(* IEC 61131-3 sources: RL_MAR/experiments/results/ablation/Ablation_single_agent_deepseek-ai_DeepSeek-V3.2_20260603_033757 (part 2) *)

(* ---- med_51.st ---- *)
FUNCTION_BLOCK PizzaMakingMachine
VAR_INPUT
    StartButton : BOOL;
    StopButton : BOOL;
    DoughReadySensor : BOOL;
    ToppingsReadySensor : BOOL;
    BakingDoneSensor : BOOL;
END_VAR

VAR_OUTPUT
    DoughRollerMotor : BOOL;
    ToppingDispenser : BOOL;
    ConveyorMotor : BOOL;
    OvenHeater : BOOL;
    OvenTemperature : INT;
END_VAR

VAR
    State : INT := 0; (* 0=Idle, 1=DoughRolling, 2=ToppingDispensing, 3=ConveyingToOven, 4=Baking, 5=Complete *)
    TargetBakingTemp : INT := 220;
    IdleTemp : INT := 0;
END_VAR

(* Main state machine *)
CASE State OF
    0: (* Idle State *)
        DoughRollerMotor := FALSE;
        ToppingDispenser := FALSE;
        ConveyorMotor := FALSE;
        OvenHeater := FALSE;
        OvenTemperature := IdleTemp;

        IF StartButton AND NOT StopButton THEN
            State := 1;
        END_IF;

    1: (* Dough Rolling State *)
        IF StopButton THEN
            State := 0;
        ELSE
            DoughRollerMotor := NOT DoughReadySensor;
            ToppingDispenser := FALSE;
            ConveyorMotor := FALSE;
            OvenHeater := FALSE;
            OvenTemperature := IdleTemp;

            IF DoughReadySensor THEN
                State := 2;
            END_IF;
        END_IF;

    2: (* Topping Dispensing State *)
        IF StopButton THEN
            State := 0;
        ELSE
            DoughRollerMotor := FALSE;
            ToppingDispenser := NOT ToppingsReadySensor;
            ConveyorMotor := FALSE;
            OvenHeater := FALSE;
            OvenTemperature := IdleTemp;

            IF ToppingsReadySensor THEN
                State := 3;
            END_IF;
        END_IF;

    3: (* Convey to Oven State *)
        IF StopButton THEN
            State := 0;
        ELSE
            DoughRollerMotor := FALSE;
            ToppingDispenser := FALSE;
            ConveyorMotor := TRUE;
            OvenHeater := TRUE;
            OvenTemperature := TargetBakingTemp;

            (* Transition to baking state - in real implementation would use timer/sensor *)
            State := 4;
        END_IF;

    4: (* Baking State *)
        IF StopButton THEN
            State := 0;
        ELSE
            DoughRollerMotor := FALSE;
            ToppingDispenser := FALSE;
            ConveyorMotor := FALSE;
            OvenHeater := TRUE;
            OvenTemperature := TargetBakingTemp;

            IF BakingDoneSensor THEN
                State := 5;
            END_IF;
        END_IF;

    5: (* Baking Complete State *)
        IF StopButton THEN
            State := 0;
        ELSE
            DoughRollerMotor := FALSE;
            ToppingDispenser := FALSE;
            ConveyorMotor := FALSE;
            OvenHeater := FALSE;
            OvenTemperature := IdleTemp;

            (* Return to idle after completion *)
            State := 0;
        END_IF;

    ELSE
        (* Error state - reset to idle *)
        State := 0;
        DoughRollerMotor := FALSE;
        ToppingDispenser := FALSE;
        ConveyorMotor := FALSE;
        OvenHeater := FALSE;
        OvenTemperature := IdleTemp;
END_CASE;
END_FUNCTION_BLOCK

(* ---- med_52.st ---- *)
FUNCTION_BLOCK TrafficManagementSystem
VAR_INPUT
    VehicleCount1 : INT;
    VehicleCount2 : INT;
    VehicleCount3 : INT;
    VehicleCount4 : INT;
END_VAR

VAR_OUTPUT
    TrafficLight1 : BOOL;
    TrafficLight2 : BOOL;
    TrafficLight3 : BOOL;
    TrafficLight4 : BOOL;
END_VAR

VAR
    // Internal variables to handle tie conditions and maintain state
    bDefaultStatePair1 : BOOL := TRUE;
    bDefaultStatePair2 : BOOL := TRUE;
END_VAR

(* Pair 1: Intersection 1 vs Intersection 2 - Independent Management *)
IF VehicleCount1 > VehicleCount2 THEN
    TrafficLight1 := TRUE;
    TrafficLight2 := FALSE;
    bDefaultStatePair1 := TRUE;  // Update default for next tie
ELSIF VehicleCount2 > VehicleCount1 THEN
    TrafficLight1 := FALSE;
    TrafficLight2 := TRUE;
    bDefaultStatePair1 := FALSE;  // Update default for next tie
ELSE
    (* If counts are equal, use alternating default logic *)
    TrafficLight1 := bDefaultStatePair1;
    TrafficLight2 := NOT bDefaultStatePair1;
    bDefaultStatePair1 := NOT bDefaultStatePair1;  // Toggle for next tie
END_IF;

(* Pair 2: Intersection 3 vs Intersection 4 - Independent Management *)
IF VehicleCount3 > VehicleCount4 THEN
    TrafficLight3 := TRUE;
    TrafficLight4 := FALSE;
    bDefaultStatePair2 := TRUE;  // Update default for next tie
ELSIF VehicleCount4 > VehicleCount3 THEN
    TrafficLight3 := FALSE;
    TrafficLight4 := TRUE;
    bDefaultStatePair2 := FALSE;  // Update default for next tie
ELSE
    (* If counts are equal, use alternating default logic *)
    TrafficLight3 := bDefaultStatePair2;
    TrafficLight4 := NOT bDefaultStatePair2;
    bDefaultStatePair2 := NOT bDefaultStatePair2;  // Toggle for next tie
END_IF;

END_FUNCTION_BLOCK

(* ---- med_53.st ---- *)
FUNCTION_BLOCK PouchMachine
VAR_INPUT
    start_machine: BOOL;
    stop_machine: BOOL;
    emergency_stop: BOOL := TRUE; (* Safety input - normally TRUE *)
    tension_sensor1: BOOL; (* Tension feedback from feeder 1 *)
    tension_sensor2: BOOL; (* Tension feedback from feeder 2 *)
    cutter_home_pos: BOOL; (* Horizontal cutter at home position *)
    cutter_vert_home: BOOL; (* Vertical cutter at home position *)
END_VAR

VAR_OUTPUT
    machine_ready: BOOL;
    feeder_running: BOOL;
    cutter_running: BOOL;
    heating_running: BOOL;
    cooling_running: BOOL;
    startup_in_progress: BOOL;
    shutdown_in_progress: BOOL;
    fault_condition: BOOL;
    fault_code: INT;
END_VAR

VAR
    startup_complete: BOOL := FALSE;
    shutdown_complete: BOOL := TRUE;
    machine_state: INT := 0;
    step_timer: TON;
    heating_stations_active: ARRAY[1..8] OF BOOL;
    cooling_stations_active: ARRAY[1..8] OF BOOL;
    feeder1_tension_ok: BOOL;
    feeder2_tension_ok: BOOL;
    winding_tension_ok: BOOL;
    horizontal_cutter_ready: BOOL;
    vertical_cutter_ready: BOOL;
    startup_step: INT := 0;
    shutdown_step: INT := 0;
    i: INT;
END_VAR

(* Initialize timers *)
step_timer(IN := FALSE, PT := T#1S);

(* Main state machine *)
IF emergency_stop THEN
    CASE machine_state OF
        (* IDLE STATE *)
        0: (* Machine stopped, ready for startup *)
            machine_ready := FALSE;
            feeder_running := FALSE;
            cutter_running := FALSE;
            heating_running := FALSE;
            cooling_running := FALSE;
            startup_in_progress := FALSE;
            shutdown_in_progress := FALSE;
            fault_condition := FALSE;
            fault_code := 0;
            startup_complete := FALSE;
            shutdown_complete := TRUE;

            (* Reset all stations *)
            FOR i := 1 TO 8 DO
                heating_stations_active[i] := FALSE;
                cooling_stations_active[i] := FALSE;
            END_FOR;

            horizontal_cutter_ready := FALSE;
            vertical_cutter_ready := FALSE;
            feeder1_tension_ok := FALSE;
            feeder2_tension_ok := FALSE;
            winding_tension_ok := FALSE;

            IF start_machine AND NOT stop_machine THEN
                machine_state := 1; (* Start startup sequence *)
                startup_step := 1;
                step_timer(IN := TRUE, PT := T#1S);
            END_IF;

        (* STARTUP SEQUENCE *)
        1: (* Startup sequence active *)
            startup_in_progress := TRUE;
            shutdown_in_progress := FALSE;

            CASE startup_step OF
                1: (* Step 1: Activate heating stations *)
                    heating_running := TRUE;
                    FOR i := 1 TO 8 DO
                        heating_stations_active[i] := TRUE;
                    END_FOR;

                    IF step_timer.Q THEN
                        step_timer(IN := FALSE, PT := T#1S);
                        startup_step := 2;
                        step_timer(IN := TRUE, PT := T#1S);
                    END_IF;

                2: (* Step 2: Activate cooling stations *)
                    cooling_running := TRUE;
                    FOR i := 1 TO 8 DO
                        cooling_stations_active[i] := TRUE;
                    END_FOR;

                    IF step_timer.Q THEN
                        step_timer(IN := FALSE, PT := T#1S);
                        startup_step := 3;
                        step_timer(IN := TRUE, PT := T#2S);
                    END_IF;

                3: (* Step 3: Start feeders and establish tension *)
                    feeder_running := TRUE;

                    (* Check tension from both feeders *)
                    feeder1_tension_ok := tension_sensor1;
                    feeder2_tension_ok := tension_sensor2;
                    winding_tension_ok := feeder1_tension_ok AND feeder2_tension_ok;

                    IF step_timer.Q THEN
                        IF winding_tension_ok THEN
                            step_timer(IN := FALSE, PT := T#1S);
                            startup_step := 4;
                            step_timer(IN := TRUE, PT := T#1S);
                        ELSE
                            (* Tension not established - fault *)
                            machine_state := 99;
                            fault_condition := TRUE;
                            fault_code := 1; (* Tension fault *)
                        END_IF;
                    END_IF;

                4: (* Step 4: Activate cutters *)
                    IF cutter_home_pos AND cutter_vert_home THEN
                        horizontal_cutter_ready := TRUE;
                        vertical_cutter_ready := TRUE;
                        cutter_running := TRUE;

                        IF step_timer.Q THEN
                            step_timer(IN := FALSE, PT := T#1S);
                            startup_step := 5;
                            step_timer(IN := TRUE, PT := T#500MS);
                        END_IF;
                    ELSE
                        (* Cutters not in home position - fault *)
                        machine_state := 99;
                        fault_condition := TRUE;
                        fault_code := 2; (* Cutter position fault *)
                    END_IF;

                5: (* Step 5: Set machine to ready state *)
                    IF step_timer.Q THEN
                        machine_ready := TRUE;
                        startup_complete := TRUE;
                        shutdown_complete := FALSE;
                        startup_in_progress := FALSE;
                        machine_state := 2; (* Running state *)
                        step_timer(IN := FALSE, PT := T#1S);
                    END_IF;
            END_CASE;

            (* Check for stop command during startup *)
            IF stop_machine THEN
                machine_state := 3; (* Go to shutdown *)
                shutdown_step := 1;
                step_timer(IN := TRUE, PT := T#1S);
            END_IF;

        (* RUNNING STATE *)
        2: (* Machine running normally *)
            (* Maintain station status *)
            heating_running := TRUE;
            cooling_running := TRUE;
            feeder_running := TRUE;
            cutter_running := TRUE;

            (* Continuously monitor tension *)
            feeder1_tension_ok := tension_sensor1;
            feeder2_tension_ok := tension_sensor2;
            winding_tension_ok := feeder1_tension_ok AND feeder2_tension_ok;

            IF NOT winding_tension_ok THEN
                machine_state := 99;
                fault_condition := TRUE;
                fault_code := 3; (* Running tension fault *)
            END_IF;

            (* Check for stop command *)
            IF stop_machine THEN
                machine_state := 3; (* Start shutdown sequence *)
                shutdown_step := 1;
                step_timer(IN := TRUE, PT := T#1S);
            END_IF;

        (* SHUTDOWN SEQUENCE *)
        3: (* Shutdown sequence active *)
            startup_in_progress := FALSE;
            shutdown_in_progress := TRUE;
            machine_ready := FALSE;

            CASE shutdown_step OF
                1: (* Step 1: Stop cutters *)
                    cutter_running := FALSE;
                    horizontal_cutter_ready := FALSE;
                    vertical_cutter_ready := FALSE;

                    IF step_timer.Q THEN
                        step_timer(IN := FALSE, PT := T#1S);
                        shutdown_step := 2;
                        step_timer(IN := TRUE, PT := T#1S);
                    END_IF;

                2: (* Step 2: Stop feeders *)
                    feeder_running := FALSE;
                    feeder1_tension_ok := FALSE;
                    feeder2_tension_ok := FALSE;
                    winding_tension_ok := FALSE;

                    IF step_timer.Q THEN
                        step_timer(IN := FALSE, PT := T#1S);
                        shutdown_step := 3;
                        step_timer(IN := TRUE, PT := T#2S);
                    END_IF;

                3: (* Step 3: Deactivate heating stations *)
                    heating_running := FALSE;
                    FOR i := 1 TO 8 DO
                        heating_stations_active[i] := FALSE;
                    END_FOR;

                    IF step_timer.Q THEN
                        step_timer(IN := FALSE, PT := T#1S);
                        shutdown_step := 4;
                        step_timer(IN := TRUE, PT := T#2S);
                    END_IF;

                4: (* Step 4: Deactivate cooling stations *)
                    cooling_running := FALSE;
                    FOR i := 1 TO 8 DO
                        cooling_stations_active[i] := FALSE;
                    END_FOR;

                    IF step_timer.Q THEN
                        step_timer(IN := FALSE, PT := T#1S);
                        shutdown_step := 5;
                        step_timer(IN := TRUE, PT := T#500MS);
                    END_IF;

                5: (* Step 5: Set machine to not-ready state *)
                    IF step_timer.Q THEN
                        startup_complete := FALSE;
                        shutdown_complete := TRUE;
                        shutdown_in_progress := FALSE;
                        machine_state := 0; (* Return to idle *)
                        step_timer(IN := FALSE, PT := T#1S);
                    END_IF;
            END_CASE;

            (* Check for start command during shutdown *)
            IF start_machine AND NOT stop_machine THEN
                (* Abort shutdown and restart *)
                machine_state := 1;
                startup_step := 1;
                step_timer(IN := TRUE, PT := T#1S);
            END_IF;

        (* FAULT STATE *)
        99: (* Fault condition *)
            machine_ready := FALSE;
            feeder_running := FALSE;
            cutter_running := FALSE;
            heating_running := FALSE;
            cooling_running := FALSE;
            startup_in_progress := FALSE;
            shutdown_in_progress := FALSE;

            (* Deactivate all stations *)
            FOR i := 1 TO 8 DO
                heating_stations_active[i] := FALSE;
                cooling_stations_active[i] := FALSE;
            END_FOR;

            (* Reset fault when emergency stop is cycled *)
            IF NOT emergency_stop THEN
                machine_state := 0;
                fault_condition := FALSE;
                fault_code := 0;
            END_IF;

    END_CASE;
ELSE
    (* Emergency stop active - force everything off *)
    machine_state := 0;
    machine_ready := FALSE;
    feeder_running := FALSE;
    cutter_running := FALSE;
    heating_running := FALSE;
    cooling_running := FALSE;
    startup_in_progress := FALSE;
    shutdown_in_progress := FALSE;
    fault_condition := FALSE;
    fault_code := 0;

    FOR i := 1 TO 8 DO
        heating_stations_active[i] := FALSE;
        cooling_stations_active[i] := FALSE;
    END_FOR;

    startup_complete := FALSE;
    shutdown_complete := TRUE;
    step_timer(IN := FALSE, PT := T#1S);
END_IF;
END_FUNCTION_BLOCK

(* ---- med_54.st ---- *)
FUNCTION_BLOCK FeedForwardControl
VAR_INPUT
    FlowRate1, FlowRate2: REAL; // Input flow rates of reactants
    MixRatio: REAL; // Desired mixing ratio (Reactant1:Reactant2)
END_VAR

VAR_OUTPUT
    OutFlowRate1, OutFlowRate2: REAL; // Output flow rates for reactants to maintain the mixing ratio
END_VAR

VAR
    MixedFlowRate: REAL; // Total mixed flow rate
    ClampedFlow1, ClampedFlow2: REAL;
    RatioPart1, RatioPart2: REAL;
    RatioSum: REAL;
END_VAR

// Limit input flow rates to allowed range 0-100
ClampedFlow1 := LIMIT(0.0, FlowRate1, 100.0);
ClampedFlow2 := LIMIT(0.0, FlowRate2, 100.0);

// Calculate total mixed flow rate
MixedFlowRate := ClampedFlow1 + ClampedFlow2;

// Calculate mixing ratio parts with error handling to prevent division by zero
RatioSum := MixRatio + 1.0;
IF RatioSum > 0.0 THEN
    RatioPart1 := MixRatio / RatioSum;
    RatioPart2 := 1.0 / RatioSum;
ELSE
    // Handle invalid ratio (MixRatio = -1.0)
    RatioPart1 := 0.0;
    RatioPart2 := 0.0;
END_IF

// Calculate output flow rates based on mixing ratio and total flow rate
OutFlowRate1 := LIMIT(0.0, MixedFlowRate * RatioPart1, 100.0);
OutFlowRate2 := LIMIT(0.0, MixedFlowRate * RatioPart2, 100.0);

END_FUNCTION_BLOCK

(* ---- med_55.st ---- *)
FUNCTION_BLOCK StateMachineControl
VAR_INPUT
    request : BOOL;
    done : BOOL;
END_VAR

VAR_OUTPUT
    listen : BOOL;
END_VAR

VAR
    state : INT := 0;
END_VAR

CASE state OF
    0: // Idle state
        listen := TRUE;
        IF request THEN
            state := 1;
            listen := FALSE;
        END_IF;

    1: // Processing state
        listen := FALSE;
        IF done THEN
            state := 0;
        END_IF;

    ELSE
        // Handle unexpected state values
        state := 0;
        listen := FALSE;
END_CASE;

END_FUNCTION_BLOCK

(* ---- med_56.st ---- *)
FUNCTION_BLOCK FB_SimpleRepeat
VAR_INPUT
    INPUT_VAR1 : INT := 2;
    INPUT_COUNTER : INT := 4;
END_VAR

VAR_OUTPUT
    OUTPUT_VAR1 : INT;
END_VAR

VAR
    COUNTER : INT;
END_VAR

METHOD Run : BOOL
VAR_INPUT
    bExecute : BOOL;
END_VAR

VAR
    nTempCounter : INT;
END_VAR

IF bExecute THEN
    OUTPUT_VAR1 := INPUT_VAR1;
    nTempCounter := INPUT_COUNTER;

    REPEAT
        OUTPUT_VAR1 := OUTPUT_VAR1 * 2;
        nTempCounter := nTempCounter - 1;
    UNTIL nTempCounter <= 0
    END_REPEAT;

    Run := TRUE;
ELSE
    Run := FALSE;
END_IF;

END_METHOD

END_FUNCTION_BLOCK

(* ---- med_57.st ---- *)
FUNCTION_BLOCK FB_CourseDifferenceControl
VAR_INPUT
    KOMPASS_GRAD : INT;
    KURS : INT;
END_VAR
VAR_OUTPUT
    KURS_DIFF : INT;
END_VAR
VAR
    tempDiff : INT;
END_VAR

// Main logic
IF KOMPASS_GRAD < 0 THEN
    KURS_DIFF := 0;
ELSE
    tempDiff := KURS - KOMPASS_GRAD;

    // Handle angle wrapping (3600 = 360 degrees * 10 for decimal precision)
    IF tempDiff > 1800 THEN
        tempDiff := tempDiff - 3600;
    ELSIF tempDiff < -1800 THEN
        tempDiff := tempDiff + 3600;
    END_IF;

    KURS_DIFF := tempDiff;
END_IF;
END_FUNCTION_BLOCK

PROGRAM MAIN
VAR
    courseControl : FB_CourseDifferenceControl;
    testKOMPASS : INT;
    testKURS : INT;
    resultDiff : INT;
END_VAR

// Example usage of the function block
courseControl(KOMPASS_GRAD := testKOMPASS, KURS := testKURS);
resultDiff := courseControl.KURS_DIFF;
END_PROGRAM

(* ---- med_58.st ---- *)
FUNCTION_BLOCK FB_ThresholdAccumulator
VAR_INPUT
    i : INT;
END_VAR

VAR_OUTPUT
    o : INT;
END_VAR

VAR
    s1 : INT;
END_VAR

// Main logic
s1 := 0; // Initialize s1 at start of each call

IF i > 0 THEN
    s1 := s1 + i; // Add i to s1 if i > 0
END_IF;

IF s1 = 42 THEN
    s1 := s1 + 8000; // Add 8000 if s1 equals 42
END_IF;

// Determine output value
IF s1 < 0 THEN
    o := 0;
ELSE
    o := s1;
END_IF;

END_FUNCTION_BLOCK

(* ---- med_59.st ---- *)
FUNCTION_BLOCK FB_ConditionalSelectAndAggregate
VAR_INPUT
    Z : INT;
END_VAR
VAR
    A_X : INT := 42;
    A_Y : INT := 333;
END_VAR
VAR_OUTPUT
    NEW_Z : INT;
END_VAR

IF A_X > Z THEN
    NEW_Z := A_Y;
ELSE
    NEW_Z := Z;
END_IF;
NEW_Z := NEW_Z + A_X + A_Y;
END_FUNCTION_BLOCK

(* ---- med_60.st ---- *)
FUNCTION_BLOCK FB_RequestHandler
VAR_INPUT
    request : BOOL;
    done : BOOL;
END_VAR

VAR_OUTPUT
    listen : BOOL;
END_VAR

VAR
    state : INT := 0;
END_VAR

CASE state OF
    0:
        IF NOT request THEN
            listen := TRUE;
            state := 0;
        ELSE
            listen := FALSE;
            state := 1;
        END_IF;

    1:
        IF NOT done THEN
            state := 1;
        ELSE
            listen := TRUE;
            state := 0;
        END_IF;
END_CASE;

END_FUNCTION_BLOCK

(* ---- med_61.st ---- *)
FUNCTION_BLOCK FB_Sum
VAR_INPUT
    maxValue : INT;
END_VAR
VAR_OUTPUT
    wData : WORD;
END_VAR

VAR
    II : INT;
END_VAR

BEGIN
    wData := 0;

    FOR II := 0 TO maxValue DO
        wData := wData + WORD(II);
    END_FOR;
END_FUNCTION_BLOCK

(* ---- med_62.st ---- *)
FUNCTION_BLOCK FB_PedestrianTrafficLight
VAR_INPUT
    pedBtnPress : BOOL;
END_VAR
VAR_OUTPUT
    carLightIsGreen : BOOL;
    pedLightIsGreen : BOOL;
    TimeCounter : INT;
END_VAR
VAR
    buttonPressedBefore : BOOL := FALSE;
    currentState : INT := 0; // 0: CarGreen, 1: CarRed_Waiting, 2: PedGreen, 3: PedRed_Waiting
END_VAR

CASE currentState OF
    0: // State 0: Car Green
        carLightIsGreen := TRUE;
        pedLightIsGreen := FALSE;
        TimeCounter := 0;

        // Check for button press transition
        IF (pedBtnPress AND NOT buttonPressedBefore) THEN
            currentState := 1;
            buttonPressedBefore := TRUE;
        ELSIF (pedBtnPress = FALSE) THEN
            buttonPressedBefore := FALSE;
        END_IF;

    1: // State 1: Car Red, Waiting for Pedestrian Green
        carLightIsGreen := FALSE;
        pedLightIsGreen := FALSE;
        TimeCounter := TimeCounter + 1;

        IF TimeCounter >= 10 THEN
            currentState := 2;
        END_IF;

        // Update button memory
        IF (pedBtnPress = FALSE) THEN
            buttonPressedBefore := FALSE;
        END_IF;

    2: // State 2: Pedestrian Green
        carLightIsGreen := FALSE;
        pedLightIsGreen := TRUE;
        TimeCounter := TimeCounter + 1;

        IF TimeCounter >= 40 THEN
            currentState := 3;
        END_IF;

        // Update button memory
        IF (pedBtnPress = FALSE) THEN
            buttonPressedBefore := FALSE;
        END_IF;

    3: // State 3: Pedestrian Red, Waiting for Car Green
        carLightIsGreen := FALSE;
        pedLightIsGreen := FALSE;
        TimeCounter := TimeCounter + 1;

        IF TimeCounter >= 50 THEN
            currentState := 0;
        END_IF;

        // Update button memory
        IF (pedBtnPress = FALSE) THEN
            buttonPressedBefore := FALSE;
        END_IF;
END_CASE;

END_FUNCTION_BLOCK

(* ---- med_63.st ---- *)
FUNCTION MoveCarToExitGate : BOOL
VAR_INPUT
    SpaceNumber : INT;
END_VAR
VAR
    // Add any necessary internal variables for movement logic
    // For example: Timer, Step counter, etc.
END_VAR

// Implement car movement logic here
// This is a placeholder - actual implementation would depend on hardware specifics
MoveCarToExitGate := TRUE; // Return TRUE when movement is complete
END_FUNCTION

FUNCTION_BLOCK Automated_Parking_Controller
VAR_INPUT
    EntryGateSensor : BOOL; (* Sensor input for entry gate *)
    ExitGateSensor : BOOL; (* Sensor input for exit gate *)
    CarDetected : BOOL; (* Sensor input for car detection *)
END_VAR
VAR_OUTPUT
    ParkingSpaceNumber : INT := 0; (* Allocated parking space number *)
    RetrievalInProgress : BOOL := FALSE; (* Flag for car retrieval in progress *)
END_VAR
VAR
    ParkingSpaces : ARRAY[1..100] OF BOOL; (* Parking space status: TRUE=Occupied, FALSE=Available *)
    i : INT; (* Loop counter *)
    SpaceToRetrieve : INT := 0; (* Parking space number for retrieval *)
    MovementComplete : BOOL; (* Flag to track movement completion *)
END_VAR

// Main program logic
IF NOT RetrievalInProgress THEN
    // Entry Gate Management
    IF EntryGateSensor THEN
        // Find first available parking space
        ParkingSpaceNumber := 0;
        FOR i := 1 TO 100 DO
            IF NOT ParkingSpaces[i] THEN
                ParkingSpaces[i] := TRUE;
                ParkingSpaceNumber := i;
                EXIT;
            END_IF;
        END_FOR;
    END_IF;

    // Exit Gate Management
    IF ExitGateSensor AND (ParkingSpaceNumber > 0) THEN
        ParkingSpaces[ParkingSpaceNumber] := FALSE;
        ParkingSpaceNumber := 0;
    END_IF;

    // Start car retrieval when detected
    IF CarDetected AND (ParkingSpaceNumber > 0) THEN
        RetrievalInProgress := TRUE;
        SpaceToRetrieve := ParkingSpaceNumber;
        MovementComplete := FALSE;
    END_IF;
END_IF;

// Car Retrieval Management
IF RetrievalInProgress THEN
    IF NOT MovementComplete THEN
        // Call the function (not instantiate it)
        MovementComplete := MoveCarToExitGate(SpaceToRetrieve);
    ELSE
        // Mark space as available and reset
        ParkingSpaces[SpaceToRetrieve] := FALSE;
        ParkingSpaceNumber := 0;
        RetrievalInProgress := FALSE;
        MovementComplete := FALSE;
        SpaceToRetrieve := 0;
    END_IF;
END_IF;
END_FUNCTION_BLOCK

(* ---- med_64.st ---- *)
FUNCTION_BLOCK BakeryOvenControl
VAR_INPUT
    TemperatureSensor : REAL;        (* Current measured oven temperature in °C *)
    HumiditySensor : REAL;           (* Current measured oven humidity in %RH *)
    StartBaking : BOOL;              (* Command to start baking cycle *)
    StopBaking : BOOL;               (* Command to stop baking cycle immediately *)
END_VAR

VAR_OUTPUT
    HeatingElement : BOOL;           (* Control signal for heating element *)
    CoolingElement : BOOL;           (* Control signal for cooling element *)
    HumidityControl : BOOL;          (* Control signal for humidification system *)
    DehumidityControl : BOOL;        (* Control signal for dehumidification system *)
    BakingComplete : BOOL;           (* Signal indicating baking cycle is complete *)
    RemainingTime : TIME;            (* Remaining baking time display *)
END_VAR

VAR
    (* Setpoints - initialized when oven is off *)
    TemperatureSetpoint : REAL := 180.0;     (* Desired baking temperature in °C *)
    HumiditySetpoint : REAL := 65.0;         (* Desired baking humidity in %RH *)
    BakingTimeSetpoint : TIME := T#30M;      (* Total baking time *)

    (* Control thresholds - configurable for different baking requirements *)
    TemperatureThreshold : REAL := 2.0;      (* Temperature deadband threshold *)
    HumidityThreshold : REAL := 5.0;         (* Humidity deadband threshold *)

    (* Internal state variables *)
    OvenActive : BOOL := FALSE;              (* TRUE when baking cycle is active *)
    TimerValue : TIME := T#0S;               (* Current timer value *)
    TimerEnable : BOOL := FALSE;             (* Timer enable flag *)

    (* Edge detection for start/stop commands *)
    StartRisingEdge : R_TRIG;
    StopRisingEdge : R_TRIG;
END_VAR

(* Edge detection for start/stop commands *)
StartRisingEdge(CLK := StartBaking);
StopRisingEdge(CLK := StopBaking);

(* Main control logic *)
IF NOT OvenActive THEN
    (* Oven is inactive - deactivate all outputs *)
    HeatingElement := FALSE;
    CoolingElement := FALSE;
    HumidityControl := FALSE;
    DehumidityControl := FALSE;
    BakingComplete := FALSE;
    TimerValue := T#0S;
    TimerEnable := FALSE;

    (* Initialize setpoints when oven is off (can be modified externally) *)
    TemperatureSetpoint := 180.0;    (* Default temperature setpoint *)
    HumiditySetpoint := 65.0;        (* Default humidity setpoint *)
    BakingTimeSetpoint := T#30M;     (* Default baking time *)

    (* Start baking cycle on rising edge of StartBaking *)
    IF StartRisingEdge.Q THEN
        OvenActive := TRUE;
        TimerValue := BakingTimeSetpoint;
        TimerEnable := TRUE;
        BakingComplete := FALSE;
    END_IF;

ELSE
    (* Oven is active - implement control logic *)

    (* Stop baking immediately if stop command received *)
    IF StopRisingEdge.Q THEN
        OvenActive := FALSE;
        HeatingElement := FALSE;
        CoolingElement := FALSE;
        HumidityControl := FALSE;
        DehumidityControl := FALSE;
        BakingComplete := TRUE;
        TimerEnable := FALSE;
    ELSE
        (* Temperature Control Logic *)
        IF TemperatureSensor < (TemperatureSetpoint - TemperatureThreshold) THEN
            (* Temperature below lower threshold - activate heating *)
            HeatingElement := TRUE;
            CoolingElement := FALSE;
        ELSIF TemperatureSensor > (TemperatureSetpoint + TemperatureThreshold) THEN
            (* Temperature above upper threshold - activate cooling *)
            HeatingElement := FALSE;
            CoolingElement := TRUE;
        ELSE
            (* Temperature within acceptable range - turn off both systems *)
            HeatingElement := FALSE;
            CoolingElement := FALSE;
        END_IF;

        (* Humidity Control Logic *)
        IF HumiditySensor < (HumiditySetpoint - HumidityThreshold) THEN
            (* Humidity below lower threshold - activate humidification *)
            HumidityControl := TRUE;
            DehumidityControl := FALSE;
        ELSIF HumiditySensor > (HumiditySetpoint + HumidityThreshold) THEN
            (* Humidity above upper threshold - activate dehumidification *)
            HumidityControl := FALSE;
            DehumidityControl := TRUE;
        ELSE
            (* Humidity within acceptable range - turn off both systems *)
            HumidityControl := FALSE;
            DehumidityControl := FALSE;
        END_IF;

        (* Baking Timer Logic *)
        IF TimerEnable AND (TimerValue > T#0S) THEN
            (* Decrement timer at one-second intervals *)
            TimerValue := TimerValue - T#1S;
        END_IF;

        (* Check if baking is complete *)
        IF TimerValue <= T#0S THEN
            (* Baking time elapsed - turn off all systems *)
            HeatingElement := FALSE;
            CoolingElement := FALSE;
            HumidityControl := FALSE;
            DehumidityControl := FALSE;
            BakingComplete := TRUE;
            TimerEnable := FALSE;
            OvenActive := FALSE;
        ELSE
            BakingComplete := FALSE;
        END_IF;
    END_IF;
END_IF;

(* Output remaining time for display *)
RemainingTime := TimerValue;

END_FUNCTION_BLOCK

(* ---- med_65.st ---- *)
FUNCTION_BLOCK TheaterControl
VAR_INPUT
    StartButton : BOOL;        (* Input for starting a performance *)
    StopButton : BOOL;         (* Input for stopping a performance *)
    SceneNumber : INT;         (* Input for selecting the scene or act *)
END_VAR
VAR_OUTPUT
    LightingControl : BOOL;    (* Output for controlling lighting *)
    SoundControl : BOOL;       (* Output for controlling sound *)
    PerformanceInProgress : BOOL; (* Indicator for an ongoing performance *)
END_VAR
VAR
    bStartRisingEdge : BOOL;   (* Edge detection for start button *)
    bPrevStartState : BOOL;    (* Previous state for edge detection *)
END_VAR

(* Edge detection for StartButton *)
bStartRisingEdge := StartButton AND NOT bPrevStartState;
bPrevStartState := StartButton;

(* Main control logic *)
IF StopButton THEN
    (* Immediate stop override *)
    LightingControl := FALSE;
    SoundControl := FALSE;
    PerformanceInProgress := FALSE;
ELSIF NOT PerformanceInProgress AND bStartRisingEdge THEN
    (* Start new performance if not already in progress *)
    IF (SceneNumber >= 1) AND (SceneNumber <= 3) THEN
        LightingControl := TRUE;
        SoundControl := TRUE;
        PerformanceInProgress := TRUE;
    ELSE
        (* Invalid scene number *)
        LightingControl := FALSE;
        SoundControl := FALSE;
        PerformanceInProgress := FALSE;
    END_IF;
ELSIF PerformanceInProgress THEN
    (* Maintain performance state *)
    IF (SceneNumber >= 1) AND (SceneNumber <= 3) THEN
        LightingControl := TRUE;
        SoundControl := TRUE;
        PerformanceInProgress := TRUE;
    ELSE
        (* Scene changed to invalid during performance - stop performance *)
        LightingControl := FALSE;
        SoundControl := FALSE;
        PerformanceInProgress := FALSE;
    END_IF;
ELSE
    (* Idle state - ensure outputs are off *)
    LightingControl := FALSE;
    SoundControl := FALSE;
    PerformanceInProgress := FALSE;
END_IF;
END_FUNCTION_BLOCK

(* ---- med_66.st ---- *)
FUNCTION_BLOCK ElevatorControl
VAR_INPUT
    CurrentPos : INT;
    RequestedPos : INT;
    ButtonPressed : BOOL;
END_VAR
VAR_OUTPUT
    MotorMovingUp : BOOL;
    MotorMovingDown : BOOL;
    DoorIsOpen : BOOL;
END_VAR
VAR
    bMoving : BOOL := FALSE;
END_VAR

(* Main elevator control logic *)
IF ButtonPressed THEN
    (* Close door when button is pressed *)
    DoorIsOpen := FALSE;

    (* Determine movement direction based on position comparison *)
    IF RequestedPos > CurrentPos THEN
        MotorMovingUp := TRUE;
        MotorMovingDown := FALSE;
        bMoving := TRUE;
    ELSIF RequestedPos < CurrentPos THEN
        MotorMovingUp := FALSE;
        MotorMovingDown := TRUE;
        bMoving := TRUE;
    ELSE
        (* Already at requested floor *)
        MotorMovingUp := FALSE;
        MotorMovingDown := FALSE;
        bMoving := FALSE;
        DoorIsOpen := TRUE;
    END_IF;
END_IF;

(* Stop and open door when reaching requested floor *)
IF CurrentPos = RequestedPos AND bMoving THEN
    MotorMovingUp := FALSE;
    MotorMovingDown := FALSE;
    bMoving := FALSE;
    DoorIsOpen := TRUE;
END_IF;

(* Ensure door remains closed while moving *)
IF bMoving THEN
    DoorIsOpen := FALSE;
END_IF;

(* Safety: Ensure motor cannot move in both directions simultaneously *)
IF MotorMovingUp AND MotorMovingDown THEN
    MotorMovingUp := FALSE;
    MotorMovingDown := FALSE;
    bMoving := FALSE;
END_IF;

END_FUNCTION_BLOCK

(* ---- med_67.st ---- *)
FUNCTION_BLOCK FB_FactorialCalculator
VAR_INPUT
    X : INT;
END_VAR

VAR_OUTPUT
    FactorialResult : INT;
    FactorialGoodResult : INT;
END_VAR

VAR
    tempGoodResult : INT;
END_VAR

// Initialize outputs
FactorialGoodResult := 0;
FactorialResult := 1;

// Check if input is within valid range
IF (X >= -3) AND (X <= 3) THEN
    // Calculate X^4 (X multiplied by itself 4 times)
    tempGoodResult := X * X * X * X;
    FactorialGoodResult := tempGoodResult;

    // Calculate FactorialResult based on FactorialGoodResult
    IF tempGoodResult > 1 THEN
        FactorialResult := tempGoodResult * (tempGoodResult - 1);
    ELSE
        FactorialResult := tempGoodResult;
    END_IF;
END_IF;

// If X is outside range [-3, 3], outputs remain at initialized values
// FactorialResult = 1 (as per overflow prevention requirement)
// FactorialGoodResult = 0
END_FUNCTION_BLOCK

(* ---- med_68.st ---- *)
FUNCTION_BLOCK FB_SignalControl
VAR_INPUT
    Int1 : BOOL;
    Int2 : BOOL;
    Int3 : BOOL;
    Int4 : BOOL;
    Int5 : BOOL;
    Int6 : BOOL;
    Int7 : BOOL;
    Int8 : BOOL;
    IntAn1 : UINT;
    IntAn2 : UINT;
    IntAn3 : UINT;
    IntAn4 : UINT;
    IntAn5 : UINT;
    IntAn6 : UINT;
    IntAn7 : UINT;
    IntAn8 : UINT;
    Marca2 : BOOL;
END_VAR

VAR_OUTPUT
    Out1 : BOOL;
    Out2 : BOOL;
    Out3 : BOOL;
    Out4 : BOOL;
    Out5 : BOOL;
    Out6 : BOOL;
    Out7 : BOOL;
    Out8 : BOOL;
    OutAn1 : UINT;
    OutAn2 : UINT;
    OutAn3 : UINT;
    OutAn4 : UINT;
    OutAn5 : UINT;
    OutAn6 : UINT;
    OutAn7 : UINT;
    OutAn8 : UINT;
END_VAR

VAR
    Marca1 : BOOL;
END_VAR

// Logic Implementation
// Marca1 and Marca2 latch logic
Marca1 := (NOT Marca2 AND (Marca1 OR NOT Out1) AND Int1) OR (Marca1 AND NOT Int1);
Marca2 := (NOT Marca1 AND (Marca2 OR Out1) AND Int1) OR (Marca2 AND NOT Int1);

// Out1 latch behavior
Out1 := (NOT Marca2 AND (Marca1 OR Out1)) OR (Out1 AND Marca2);

// Direct Boolean pass-through
Out2 := Int2;
Out3 := Int3;
Out4 := Int4;

// Direct unsigned integer pass-through
OutAn1 := IntAn1;
OutAn2 := IntAn2;
OutAn3 := IntAn3;
OutAn4 := IntAn4;

// Conditional output logic for Out5 to Out8
Out5 := (IntAn5 > 1000) AND NOT Int5;
Out6 := (IntAn6 > 1000) AND NOT Int6;
Out7 := (IntAn7 > 1000) AND NOT Int7;
Out8 := (IntAn8 > 1000) AND NOT Int8;

// Analog outputs pass-through for IntAn5 to IntAn8
OutAn5 := IntAn5;
OutAn6 := IntAn6;
OutAn7 := IntAn7;
OutAn8 := IntAn8;

END_FUNCTION_BLOCK

(* ---- med_69.st ---- *)
FUNCTION_BLOCK FB_ValueOut
VAR_INPUT
    valueIn : INT;
    conf : UINT;
END_VAR

VAR_OUTPUT
    ValueOut : INT;
END_VAR

VAR
END_VAR

METHOD ProcessValue : INT
VAR_INPUT
    valueIn : INT;
    conf : UINT;
END_VAR
VAR_OUTPUT
    result : INT;
END_VAR
BEGIN
    result := 0;

    CASE conf OF
        1, 2:
            IF valueIn <> 0 THEN
                result := valueIn / 10;
            END_IF;

        3:
            CASE valueIn OF
                0:   result := 0;
                300: result := 163;
                600: result := 331;
            ELSE
                result := 0;
            END_CASE;

        6, 7:
            IF valueIn = 100 THEN
                result := 319;
            ELSE
                result := 0;
            END_IF;

    ELSE
        result := 0;
    END_CASE;

    // Ensure non-negative output
    IF result < 0 THEN
        result := 0;
    END_IF;

    RETURN result;
END_METHOD

BEGIN
    ValueOut := ProcessValue(valueIn := valueIn, conf := conf);
END_FUNCTION_BLOCK

(* ---- med_70.st ---- *)
FUNCTION_BLOCK EggIncubatorControl
VAR_INPUT
    StartButton : BOOL;           (* Input for starting the incubation process *)
    StopButton : BOOL;            (* Input for stopping the incubation process *)
    TemperatureSensor : REAL;     (* Input for temperature reading in °C *)
    HumiditySensor : REAL;        (* Input for humidity reading in % *)
END_VAR
VAR_OUTPUT
    HeatingElement : BOOL;        (* Output for controlling the heating element *)
    Humidifier : BOOL;            (* Output for controlling the humidifier *)
    EggTurningMotor : BOOL;       (* Output for controlling the egg turning motor *)
    IncubationInProgress : BOOL;  (* Indicator for an ongoing incubation process *)
END_VAR
VAR
    TargetTemperature : REAL;     (* Target temperature in °C *)
    TargetHumidity : REAL;        (* Target humidity in % *)
    TurnIntervalSeconds : INT;    (* Interval for turning eggs (1 hour in seconds) *)
    TurnTimerSeconds : INT;       (* Timer for egg turning cycle in seconds *)
    MotorToggleFlag : BOOL;       (* Flag to track motor toggle state *)
END_VAR

(* Initialization of control parameters *)
TargetTemperature := 37.5;
TargetHumidity := 50.0;
TurnIntervalSeconds := 3600;

(* Start/Stop Control *)
IF StopButton THEN
    IncubationInProgress := FALSE;
    HeatingElement := FALSE;
    Humidifier := FALSE;
    EggTurningMotor := FALSE;
    TurnTimerSeconds := 0;
    MotorToggleFlag := FALSE;
ELSIF StartButton AND NOT IncubationInProgress THEN
    IncubationInProgress := TRUE;
    TurnTimerSeconds := 0;
    MotorToggleFlag := FALSE;
END_IF;

(* Temperature Control *)
IF IncubationInProgress THEN
    HeatingElement := (TemperatureSensor < TargetTemperature);
ELSE
    HeatingElement := FALSE;
END_IF;

(* Humidity Control *)
IF IncubationInProgress THEN
    Humidifier := (HumiditySensor < TargetHumidity);
ELSE
    Humidifier := FALSE;
END_IF;

(* Egg Turning Cycle *)
IF IncubationInProgress THEN
    TurnTimerSeconds := TurnTimerSeconds + 1;

    IF TurnTimerSeconds >= TurnIntervalSeconds THEN
        MotorToggleFlag := NOT MotorToggleFlag;
        EggTurningMotor := MotorToggleFlag;
        TurnTimerSeconds := 0;
    END_IF;
ELSE
    EggTurningMotor := FALSE;
    TurnTimerSeconds := 0;
END_IF;

END_FUNCTION_BLOCK

(* ---- med_71.st ---- *)
FUNCTION_BLOCK FB_Fibonacci_Calculator
VAR_INPUT
    N : DINT := 5;
END_VAR
VAR_OUTPUT
    O : DINT := 1;
END_VAR
VAR
    F1 : DINT := 1;
    F2 : DINT := 1;
    CNT : DINT := 2;
    Temp : DINT;
END_VAR

// Handle edge cases and calculate Fibonacci with saturation
IF N <= 0 THEN
    O := 0;
ELSIF N <= 2 THEN
    O := 1;
ELSE
    // Initialize Fibonacci sequence
    F1 := 1;
    F2 := 1;
    CNT := 2;

    // Calculate Fibonacci numbers up to N-th term
    WHILE CNT < N DO
        // Calculate next Fibonacci number with saturation check
        Temp := F1 + F2;

        // Apply saturation arithmetic - limit to INT maximum (32767)
        IF Temp > 32767 THEN
            Temp := 32767;
        END_IF;

        // Shift values for next iteration
        F1 := F2;
        F2 := Temp;

        // Increment counter
        CNT := CNT + 1;
    END_WHILE;

    // Output the N-th Fibonacci number
    O := F2;
END_IF;
END_FUNCTION_BLOCK

(* ---- med_72.st ---- *)
FUNCTION_BLOCK DigitalSignageManagement
VAR_INPUT
    DisplayLocations : ARRAY[1..10] OF BOOL;    (* Display status at each location *)
    ContentSource : ARRAY[1..10] OF INT;        (* Desired content for each location *)
END_VAR
VAR_OUTPUT
    CurrentContent : ARRAY[1..10] OF INT;       (* Current displayed content *)
END_VAR
VAR
    i : INT;                                    (* Loop counter *)
END_VAR

(* Main logic: Update content immediately based on inputs *)
FOR i := 1 TO 10 DO
    IF DisplayLocations[i] THEN
        (* Check if content code is valid (1, 2, or 3) *)
        CASE ContentSource[i] OF
            1: CurrentContent[i] := 1;    (* News *)
            2: CurrentContent[i] := 2;    (* Weather *)
            3: CurrentContent[i] := 3;    (* Promotional Content *)
        ELSE
            CurrentContent[i] := 0;       (* Invalid code or 0 = No Content *)
        END_CASE;
    ELSE
        (* Display is offline *)
        CurrentContent[i] := 0;
    END_IF;
END_FOR;

END_FUNCTION_BLOCK

(* ---- med_73.st ---- *)
FUNCTION_BLOCK RoboticWeldingSystem
VAR_INPUT
    RobotArm1Ready : BOOL;    (* Input for robot arm 1 ready status *)
    RobotArm2Ready : BOOL;    (* Input for robot arm 2 ready status *)
    WeldingGunReady : BOOL;   (* Input for welding gun ready status *)
    StartButton : BOOL;       (* Input for start button press *)
    StopButton : BOOL;        (* Input for stop button press *)
END_VAR
VAR_OUTPUT
    WeldingTrigger : BOOL;    (* Output to trigger welding *)
    WeldingComplete : BOOL;   (* Output indicating welding completion *)
END_VAR
VAR
    eState : (IDLE, WELDING); (* State variable for process control *)
END_VAR

(* Main state machine logic *)
CASE eState OF
    IDLE:
        WeldingTrigger := FALSE;
        WeldingComplete := TRUE;

        IF StopButton THEN
            (* Safety stop pressed - remain in IDLE *)
            eState := IDLE;
            WeldingComplete := TRUE;
        ELSIF RobotArm1Ready AND RobotArm2Ready AND WeldingGunReady AND StartButton THEN
            (* All conditions met - start welding *)
            eState := WELDING;
            WeldingComplete := FALSE;
        END_IF;

    WELDING:
        WeldingTrigger := TRUE;
        WeldingComplete := FALSE;

        IF StopButton THEN
            (* Safety stop pressed - abort welding *)
            eState := IDLE;
            WeldingTrigger := FALSE;
            WeldingComplete := TRUE;
        END_IF;
END_CASE;
END_FUNCTION_BLOCK

(* ---- med_74.st ---- *)
FUNCTION_BLOCK TrafficManagementSystem
VAR_INPUT
    VehicleCount1 : INT; (* Input for vehicle count at intersection 1 *)
    VehicleCount2 : INT; (* Input for vehicle count at intersection 2 *)
    VehicleCount3 : INT; (* Input for vehicle count at intersection 3 *)
    VehicleCount4 : INT; (* Input for vehicle count at intersection 4 *)
END_VAR
VAR_OUTPUT
    TrafficLight1 : BOOL; (* Output for traffic light at intersection 1 *)
    TrafficLight2 : BOOL; (* Output for traffic light at intersection 2 *)
    TrafficLight3 : BOOL; (* Output for traffic light at intersection 3 *)
    TrafficLight4 : BOOL; (* Output for traffic light at intersection 4 *)
END_VAR

(* Main logic *)
TrafficLight1 := (VehicleCount1 > VehicleCount2);
TrafficLight2 := NOT TrafficLight1;
TrafficLight3 := (VehicleCount3 > VehicleCount4);
TrafficLight4 := NOT TrafficLight3;

END_FUNCTION_BLOCK

(* ---- med_75.st ---- *)
FUNCTION_BLOCK HomeBrewingSystem
VAR_INPUT
    TemperatureSensor : REAL;      (* Current temperature in °C *)
    WaterFlowSensor : REAL;        (* Current water flow in L/min *)
    BrewingStartTime : TIME;       (* Start time of brewing process *)
    BrewingDuration : TIME;        (* Total brewing duration *)
END_VAR
VAR_OUTPUT
    HeatingElement : BOOL;         (* Control signal for heating element *)
    AgitationMotor : BOOL;         (* Control signal for agitation motor *)
    HopsDispenser : BOOL;          (* Control signal for hops dispenser *)
    FermentationTank : BOOL;       (* Control signal for fermentation tank transfer *)
END_VAR
VAR
    CurrentTime : TIME;            (* Current system time *)
    ElapsedBrewingTime : TIME;     (* Time elapsed since brewing start *)
    HopsDispensed : BOOL;          (* Flag to track if hops have been dispensed *)
    TankTransferred : BOOL;        (* Flag to track if transfer to fermentation tank occurred *)
END_VAR

(* Get current time *)
CurrentTime := TIME();

(* Calculate elapsed brewing time *)
ElapsedBrewingTime := CurrentTime - BrewingStartTime;

(* Temperature control logic *)
IF TemperatureSensor < 65.0 THEN
    HeatingElement := TRUE;
ELSE
    HeatingElement := FALSE;
END_IF;

(* Water flow control logic *)
IF WaterFlowSensor > 0.5 THEN
    AgitationMotor := TRUE;
ELSE
    AgitationMotor := FALSE;
END_IF;

(* Hops dispensing logic - dispense once after 5 hours *)
IF (ElapsedBrewingTime >= T#5h) AND (ElapsedBrewingTime <= BrewingDuration) AND NOT HopsDispensed THEN
    HopsDispenser := TRUE;
    HopsDispensed := TRUE;
ELSE
    HopsDispenser := FALSE;
END_IF;

(* Fermentation tank transfer logic - transfer once after 48 hours *)
IF (ElapsedBrewingTime >= T#48h) AND (ElapsedBrewingTime <= BrewingDuration) AND NOT TankTransferred THEN
    FermentationTank := TRUE;
    TankTransferred := TRUE;
ELSE
    FermentationTank := FALSE;
END_IF;

(* Reset flags when brewing duration is exceeded or before new brew starts *)
IF (ElapsedBrewingTime > BrewingDuration) OR (ElapsedBrewingTime < T#0s) THEN
    HopsDispensed := FALSE;
    TankTransferred := FALSE;
END_IF;

END_FUNCTION_BLOCK

(* ---- med_76.st ---- *)
FUNCTION_BLOCK MultimediaArtInstallationControl
VAR_INPUT
    MotionSensor : BOOL; (* Motion detection input *)
    AudioTrack : BOOL; (* Selected audio track *)
    VisualContent : BOOL; (* Selected visual content *)
END_VAR

VAR_OUTPUT
    LightingControl : BOOL; (* Lighting control output *)
    AudioControl : BOOL; (* Audio playback control *)
    VisualControl : BOOL; (* Visual display control *)
    ActivationTimer : INT; (* Timer for activation duration *)
END_VAR

VAR
    bMotionDetectedPrev : BOOL; (* Previous state of motion sensor for edge detection *)
    bElementsActive : BOOL; (* Flag indicating if elements are currently active *)
    tActivationTime : TIME; (* Activation time accumulator *)
    tNoMotionTime : TIME; (* No motion time accumulator *)
    bSafetyCheckOK : BOOL; (* Safety check status *)
END_VAR

VAR CONSTANT
    MAX_ACTIVATION_TIME : TIME := T#300S; (* Maximum activation time: 300 seconds *)
    DEBOUNCE_TIME : TIME := T#500MS; (* Debounce time for motion sensor *)
    SAFETY_CHECK_INTERVAL : TIME := T#10S; (* Interval for safety checks *)
END_VAR

(* Main control logic *)
IF NOT bSafetyCheckOK THEN
    (* Safety check failed - deactivate all elements *)
    LightingControl := FALSE;
    AudioControl := FALSE;
    VisualControl := FALSE;
    ActivationTimer := 0;
    tActivationTime := T#0S;
    tNoMotionTime := T#0S;
    bElementsActive := FALSE;
ELSE
    (* Edge detection for motion sensor with debouncing *)
    IF MotionSensor AND NOT bMotionDetectedPrev THEN
        (* Rising edge detected - start debounce timer *)
        tNoMotionTime := T#0S;
    ELSIF NOT MotionSensor AND bMotionDetectedPrev THEN
        (* Falling edge detected - start debounce timer *)
        tNoMotionTime := T#0S;
    END_IF;

    (* Update previous state *)
    bMotionDetectedPrev := MotionSensor;

    (* Check if motion is consistently detected for debounce time *)
    IF MotionSensor AND (tNoMotionTime >= DEBOUNCE_TIME) THEN
        (* Valid motion detected - activate elements *)
        IF NOT bElementsActive THEN
            (* Only activate if elements were not already active *)
            bElementsActive := TRUE;
            tActivationTime := T#0S;
        END_IF;
    ELSIF NOT MotionSensor AND (tNoMotionTime >= DEBOUNCE_TIME) THEN
        (* No motion detected for debounce time - deactivate elements *)
        bElementsActive := FALSE;
        tActivationTime := T#0S;
    END_IF;

    (* Control multimedia elements based on activation state and safety *)
    IF bElementsActive AND (tActivationTime < MAX_ACTIVATION_TIME) THEN
        (* Activate all elements *)
        LightingControl := TRUE;
        AudioControl := AudioTrack; (* Only activate if audio track is selected *)
        VisualControl := VisualContent; (* Only activate if visual content is selected *)

        (* Increment activation timer *)
        tActivationTime := tActivationTime + T#1S;
        ActivationTimer := TIME_TO_INT(tActivationTime);
    ELSE
        (* Deactivate all elements *)
        LightingControl := FALSE;
        AudioControl := FALSE;
        VisualControl := FALSE;

        (* Reset timer if elements are not active *)
        IF NOT bElementsActive THEN
            ActivationTimer := 0;
            tActivationTime := T#0S;
        END_IF;
    END_IF;

    (* Increment no motion timer when no motion is detected *)
    IF NOT MotionSensor THEN
        tNoMotionTime := tNoMotionTime + T#1S;
    ELSE
        tNoMotionTime := T#0S;
    END_IF;

    (* Safety protocol: Check power usage and system status *)
    (* This is a placeholder for actual safety checks *)
    bSafetyCheckOK := TRUE; (* Replace with actual safety logic *)

    (* Additional safety: Force deactivation if maximum time reached *)
    IF tActivationTime >= MAX_ACTIVATION_TIME THEN
        bElementsActive := FALSE;
        LightingControl := FALSE;
        AudioControl := FALSE;
        VisualControl := FALSE;
    END_IF;
END_IF;
END_FUNCTION_BLOCK

(* ---- med_77.st ---- *)
FUNCTION_BLOCK OutdoorLEDLightingControl
VAR_INPUT
    AmbientLight : REAL;    (* Ambient light sensor input in Lux *)
    MotionSensor : BOOL;    (* Motion sensor input *)
    EnergySaving : BOOL;    (* Energy saving mode switch *)
END_VAR

VAR_OUTPUT
    Light : BOOL;           (* LED lighting control output *)
    EnergyMode : BOOL;      (* Energy saving mode status output *)
END_VAR

(* Main control logic *)
IF MotionSensor THEN
    (* Motion Detection Override *)
    Light := TRUE;
    EnergyMode := FALSE;    (* Override energy-saving mode *)
ELSE
    (* No motion detected *)
    EnergyMode := EnergySaving;    (* Reflect energy saving input *)

    (* Ambient Light and Energy Saving Control *)
    IF (AmbientLight < 50.0) AND (NOT EnergySaving) THEN
        Light := TRUE;
    ELSE
        Light := FALSE;
    END_IF;
END_IF;

END_FUNCTION_BLOCK

(* ---- med_78.st ---- *)
FUNCTION_BLOCK RetractableRoofControl
VAR_INPUT
    RainSensor : BOOL;           (* TRUE if rain is detected *)
    WindSensor : BOOL;           (* TRUE if strong wind is detected *)
    TemperatureSensor : REAL;    (* Current temperature in degrees *)
END_VAR
VAR_OUTPUT
    RoofMotor : BOOL;            (* TRUE closes roof, FALSE opens roof *)
END_VAR

(* Main control logic *)
IF RainSensor AND WindSensor THEN
    (* Combined rain and wind - highest priority *)
    RoofMotor := TRUE;
ELSIF RainSensor THEN
    (* Rain only - medium priority *)
    RoofMotor := TRUE;
ELSIF TemperatureSensor < 20.0 THEN
    (* Low temperature - lowest priority *)
    RoofMotor := TRUE;
ELSE
    (* Normal conditions - open roof *)
    RoofMotor := FALSE;
END_IF;

END_FUNCTION_BLOCK

(* ---- med_79.st ---- *)
FUNCTION_BLOCK CapsuleFillingMachineControl
VAR_INPUT
    CapsuleWeight : REAL;           // Current capsule weight
    TargetWeight : REAL;            // Target weight to achieve
    CapsuleInPosition : BOOL;       // Capsule position sensor
    HopperEmpty : BOOL;             // Hopper empty sensor
END_VAR

VAR_OUTPUT
    FeederMotor : BOOL;             // Feeder motor control
    FillingMotor : BOOL;            // Filling motor control
    ConveyorMotor : BOOL;           // Conveyor motor control
    FillingInProgress : BOOL;       // Filling status
    ErrorCode : INT;                // Error code (0=No error)
END_VAR

VAR
    // State machine
    CurrentState : INT := 0;        // 0=IDLE, 1=CONVEYING, 2=FILLING, 3=CONVEYING_OUT
    PreviousState : INT := 0;

    // Timers
    ConveyorTimer : TON;
    FillingTimer : TON;
    ConveyOutTimer : TON;
    CapsuleDetectionTimer : TON;

    // PID controller variables (simplified implementation)
    PID_Kp : REAL := 0.5;           // Proportional gain
    PID_Ki : REAL := 0.1;           // Integral gain
    PID_Kd : REAL := 0.05;          // Derivative gain
    PID_Integral : REAL := 0.0;
    PID_PreviousError : REAL := 0.0;
    PID_LastTime : REAL := 0.0;
    PID_CycleTime : REAL := 0.1;    // 100ms cycle time
    PID_Output : REAL := 0.0;

    // Control variables
    WeightTolerance : REAL := 0.1;  // Tolerance for weight comparison
    ConveyorTimeSet : TIME := T#2S; // Conveyor operation time
    FillingTimeout : TIME := T#10S; // Maximum filling time
    ConveyOutTime : TIME := T#1S;   // Convey out time
    CapsuleDetectionTimeout : TIME := T#5S; // Timeout for capsule detection

    // Internal flags
    CapsuleDetected : BOOL := FALSE;
    FillingComplete : BOOL := FALSE;
    ConveyorStarted : BOOL := FALSE;

    // Error handling
    ErrorCapsuleTimeout : BOOL := FALSE;
    ErrorFillingTimeout : BOOL := FALSE;
    ErrorHopperLow : BOOL := FALSE;

    // Temporary variables
    CurrentTime : REAL;
    Error : REAL;
    Derivative : REAL;
    dt : REAL;
END_VAR

// Initialize outputs
FeederMotor := FALSE;
FillingMotor := FALSE;
ConveyorMotor := FALSE;
FillingInProgress := FALSE;
ErrorCode := 0;

// Safety Check - Hopper Empty
IF HopperEmpty THEN
    FeederMotor := FALSE;
    FillingMotor := FALSE;
    ConveyorMotor := FALSE;
    FillingInProgress := FALSE;
    ErrorCode := 1; // Hopper empty error
    CurrentState := 0; // Return to IDLE
    RETURN;
END_IF

// Weight Validation - Initial Check
IF CapsuleWeight >= TargetWeight - WeightTolerance THEN
    FeederMotor := FALSE;
    FillingMotor := FALSE;
    ConveyorMotor := FALSE;
    FillingInProgress := FALSE;
    CurrentState := 0; // Return to IDLE
    RETURN;
END_IF

// State Machine Implementation
CASE CurrentState OF
    0: // IDLE State
        FeederMotor := FALSE;
        FillingMotor := FALSE;
        ConveyorMotor := FALSE;
        FillingInProgress := FALSE;

        // Reset timers
        ConveyorTimer(IN:=FALSE, PT:=ConveyorTimeSet);
        FillingTimer(IN:=FALSE, PT:=FillingTimeout);
        ConveyOutTimer(IN:=FALSE, PT:=ConveyOutTime);
        CapsuleDetectionTimer(IN:=FALSE, PT:=CapsuleDetectionTimeout);

        // Reset flags
        CapsuleDetected := FALSE;
        FillingComplete := FALSE;
        ConveyorStarted := FALSE;
        ErrorCapsuleTimeout := FALSE;
        ErrorFillingTimeout := FALSE;

        // Reset PID controller
        PID_Integral := 0.0;
        PID_PreviousError := 0.0;
        PID_Output := 0.0;

        // Transition to CONVEYING when capsule is detected
        IF CapsuleInPosition THEN
            CurrentState := 1;
            CapsuleDetectionTimer(IN:=TRUE, PT:=CapsuleDetectionTimeout);
        END_IF

    1: // CONVEYING State
        ConveyorMotor := TRUE;
        ConveyorStarted := TRUE;
        FillingInProgress := FALSE;

        // Start conveyor timer
        ConveyorTimer(IN:=TRUE, PT:=ConveyorTimeSet);

        // Check for capsule detection timeout
        CapsuleDetectionTimer(IN:=TRUE, PT:=CapsuleDetectionTimeout);
        IF CapsuleDetectionTimer.Q THEN
            ErrorCapsuleTimeout := TRUE;
            ErrorCode := 2; // Capsule detection timeout
            CurrentState := 0; // Return to IDLE
        END_IF

        // Transition to FILLING after conveyor time or when weight indicates capsule is in position
        IF ConveyorTimer.Q OR (CapsuleWeight > 0.1) THEN
            CurrentState := 2;
            ConveyorMotor := FALSE;
            FillingInProgress := TRUE;
            PID_LastTime := REAL_TO_TIME(T#0ms) / 1000000.0; // Initialize time
        END_IF

    2: // FILLING State
        ConveyorMotor := FALSE;
        FillingInProgress := TRUE;

        // Start filling timer
        FillingTimer(IN:=TRUE, PT:=FillingTimeout);

        // Check for filling timeout
        IF FillingTimer.Q THEN
            ErrorFillingTimeout := TRUE;
            ErrorCode := 3; // Filling timeout
            CurrentState := 0; // Return to IDLE
            FillingMotor := FALSE;
        ELSE
            // Simplified PID Controller Implementation
            CurrentTime := REAL_TO_TIME(T#0ms) / 1000000.0; // Get current time in seconds

            // Calculate time difference
            dt := CurrentTime - PID_LastTime;
            IF dt < PID_CycleTime THEN
                // Wait for next cycle
                FillingMotor := FillingMotor; // Maintain current state
            ELSE
                // Calculate error
                Error := TargetWeight - CapsuleWeight;

                // Proportional term
                PID_Output := PID_Kp * Error;

                // Integral term (with anti-windup)
                IF ABS(Error) < TargetWeight * 0.5 THEN // Only integrate when error is reasonable
                    PID_Integral := PID_Integral + (PID_Ki * Error * dt);
                    // Limit integral term
                    IF PID_Integral > 100.0 THEN
                        PID_Integral := 100.0;
                    ELSIF PID_Integral < -100.0 THEN
                        PID_Integral := -100.0;
                    END_IF;
                END_IF;

                // Derivative term
                Derivative := PID_Kd * (Error - PID_PreviousError) / dt;

                // Calculate total output
                PID_Output := PID_Output + PID_Integral + Derivative;

                // Limit output to 0-100%
                IF PID_Output > 100.0 THEN
                    PID_Output := 100.0;
                ELSIF PID_Output < 0.0 THEN
                    PID_Output := 0.0;
                END_IF;

                // Control filling motor based on PID output
                FillingMotor := (PID_Output > 5.0); // Minimum 5% output to start motor

                // Update previous values
                PID_PreviousError := Error;
                PID_LastTime := CurrentTime;
            END_IF;

            // Check if target weight is reached
            IF CapsuleWeight >= TargetWeight - WeightTolerance THEN
                FillingMotor := FALSE;
                FillingComplete := TRUE;
                CurrentState := 3; // Transition to CONVEYING_OUT
                ConveyOutTimer(IN:=TRUE, PT:=ConveyOutTime);
            END_IF;
        END_IF;

    3: // CONVEYING_OUT State
        FillingMotor := FALSE;
        ConveyorMotor := TRUE;
        FillingInProgress := FALSE;

        // Start convey out timer
        ConveyOutTimer(IN:=TRUE, PT:=ConveyOutTime);

        // Transition back to IDLE after convey out time
        IF ConveyOutTimer.Q THEN
            ConveyorMotor := FALSE;
            CurrentState := 0;
        END_IF;

    ELSE
        // Default case - return to IDLE
        CurrentState := 0;
END_CASE;

// Update error code based on error flags
IF ErrorCapsuleTimeout THEN
    ErrorCode := 2;
ELSIF ErrorFillingTimeout THEN
    ErrorCode := 3;
ELSIF ErrorHopperLow THEN
    ErrorCode := 4;
END_IF;

// Update previous state
PreviousState := CurrentState;
END_FUNCTION_BLOCK

(* ---- med_80.st ---- *)
FUNCTION_BLOCK DoughMixerControl
VAR_INPUT
    IngredientsDetected : BOOL; (* Signal indicating presence of ingredients *)
END_VAR
VAR_OUTPUT
    MixingInProgress : BOOL; (* Control signal for mixer motor *)
END_VAR
VAR
    MixingTimeElapsed : TIME; (* Current elapsed mixing time *)
    MixingTimeLimit : TIME := T#5S; (* Configurable mixing time limit *)
    PrevIngredientsDetected : BOOL; (* Previous state for edge detection *)
END_VAR

(* Main control logic *)
IF IngredientsDetected AND NOT PrevIngredientsDetected THEN
    (* Rising edge detected - start new mixing cycle *)
    MixingTimeElapsed := T#0S;
    MixingInProgress := TRUE;
ELSIF NOT IngredientsDetected OR MixingTimeElapsed >= MixingTimeLimit THEN
    (* Stop mixing if ingredients removed or time limit reached *)
    MixingInProgress := FALSE;
END_IF

(* Timer increment logic - only while mixing is active *)
IF MixingInProgress THEN
    MixingTimeElapsed := MixingTimeElapsed + T#1S;
END_IF

(* Store current state for next cycle's edge detection *)
PrevIngredientsDetected := IngredientsDetected;
END_FUNCTION_BLOCK

(* ---- med_81.st ---- *)
FUNCTION_BLOCK SolarPanelTracking
VAR
    PanelAngle : REAL; (* Output for adjusting the solar panel angle *)
    SunriseTime : TIME := T#6H; (* Set the time for sunrise (6:00 AM) *)
    SunsetTime : TIME := T#18H; (* Set the time for sunset (6:00 PM) *)
    NoonTime : TIME := T#12H; (* Set the time for solar noon (12:00 PM) *)
    MorningAngle : REAL := 30.0; (* Set the morning angle for panels *)
    NoonAngle : REAL := 60.0; (* Set the noon angle for panels *)
    EveningAngle : REAL := 30.0; (* Set the evening angle for panels *)
END_VAR
VAR_INPUT
    CurrentTime : TIME;
    SolarIntensity : REAL;
END_VAR

(* Main execution logic *)
IF SolarIntensity >= 90.0 THEN
    PanelAngle := NoonAngle;
ELSE
    IF (CurrentTime < SunriseTime) OR (CurrentTime >= SunsetTime) THEN
        PanelAngle := 0.0;
    ELSIF (CurrentTime >= SunriseTime) AND (CurrentTime < NoonTime) THEN
        PanelAngle := MorningAngle;
    ELSIF (CurrentTime >= NoonTime) AND (CurrentTime < SunsetTime) THEN
        PanelAngle := EveningAngle;
    ELSE
        PanelAngle := 0.0; (* Fallback for any unhandled time condition *)
    END_IF;
END_IF;

END_FUNCTION_BLOCK

(* ---- med_82.st ---- *)
FUNCTION_BLOCK PetFeederControl
VAR_INPUT
    CurrentTime : TIME; (* Current system time input *)
END_VAR
VAR_OUTPUT
    FoodDispense : BOOL; (* Food dispenser control signal *)
END_VAR
VAR
    FeedTime1 : TIME := T#8H0M0S; (* First feeding time - 8:00 AM *)
    FeedTime2 : TIME := T#12H0M0S; (* Second feeding time - 12:00 PM *)
    FeedTime3 : TIME := T#18H0M0S; (* Third feeding time - 6:00 PM *)
    FoodAmount : INT := 50; (* Amount of food to dispense in grams - currently unused *)
END_VAR

(* Main dispensing logic *)
FoodDispense := FALSE;

IF (CurrentTime >= FeedTime1) AND (CurrentTime < (FeedTime1 + T#30S)) THEN
    FoodDispense := TRUE;
ELSIF (CurrentTime >= FeedTime2) AND (CurrentTime < (FeedTime2 + T#30S)) THEN
    FoodDispense := TRUE;
ELSIF (CurrentTime >= FeedTime3) AND (CurrentTime < (FeedTime3 + T#30S)) THEN
    FoodDispense := TRUE;
END_IF;

END_FUNCTION_BLOCK

(* ---- med_83.st ---- *)
FUNCTION_BLOCK AmusementRideControl
VAR_INPUT
    StartButton : BOOL;        (* Start button input *)
    StopButton : BOOL;         (* Emergency stop button input *)
    SpeedSensor : REAL;        (* Speed sensor input (RPM) *)
    SafetySensor : BOOL;       (* Safety sensor status *)
END_VAR
VAR_OUTPUT
    MotorOn : BOOL := FALSE;   (* Motor control output *)
    BrakeOn : BOOL := TRUE;    (* Brake control output *)
END_VAR
VAR
    SpeedLimit : REAL := 60.0; (* Maximum allowed speed in RPM *)
END_VAR

(* Emergency Stop - Highest Priority *)
IF StopButton THEN
    MotorOn := FALSE;
    BrakeOn := TRUE;
ELSE
    (* Start Condition - All Conditions Must Be Met *)
    IF StartButton AND
       (NOT StopButton) AND
       (SpeedSensor <= SpeedLimit) AND
       SafetySensor THEN
        MotorOn := TRUE;
        BrakeOn := FALSE;
    ELSE
        MotorOn := FALSE;
        BrakeOn := TRUE;
    END_IF;

    (* Normal Operation Monitoring - Continuous Check *)
    IF MotorOn AND
       ((SpeedSensor > SpeedLimit) OR (NOT SafetySensor)) THEN
        MotorOn := FALSE;
        BrakeOn := TRUE;
    END_IF;
END_IF;

END_FUNCTION_BLOCK

(* ---- med_84.st ---- *)
FUNCTION_BLOCK ParcelSortingSystem
VAR_INPUT
    ParcelSizeSensor : REAL;           (* Sensor input for parcel size in centimeters *)
    DestinationCodeSensor : INT;       (* Destination code: 1=Location A, 2=Location B *)
END_VAR

VAR_OUTPUT
    ConveyorBeltMotor : BOOL;          (* Output for conveyor belt motor: TRUE=On, FALSE=Off *)
    SortingGate1 : BOOL;               (* Output for sorting gate 1: TRUE=Open, FALSE=Closed *)
    SortingGate2 : BOOL;               (* Output for sorting gate 2: TRUE=Open, FALSE=Closed *)
END_VAR

VAR
    SizeThreshold : REAL := 50.0;      (* Threshold to distinguish large vs small parcels *)
    MinValidSize : REAL := 5.0;        (* Minimum valid parcel size to prevent false positives *)
    MaxValidSize : REAL := 200.0;      (* Maximum valid parcel size for system capacity *)
    ValidSizeDetected : BOOL;          (* Flag indicating if parcel size is within valid range *)
    ValidDestinationDetected : BOOL;   (* Flag indicating if destination code is valid *)
END_VAR

(* Main execution logic - runs on every PLC scan cycle *)

(* Validate sensor inputs *)
ValidSizeDetected := (ParcelSizeSensor >= MinValidSize) AND (ParcelSizeSensor <= MaxValidSize);
ValidDestinationDetected := (DestinationCodeSensor = 1) OR (DestinationCodeSensor = 2);

(* Control logic based on validated inputs *)
IF ValidSizeDetected AND ValidDestinationDetected THEN
    (* Valid parcel detected - activate conveyor belt *)
    ConveyorBeltMotor := TRUE;

    (* Sorting decision logic *)
    IF ParcelSizeSensor >= SizeThreshold THEN
        (* Large parcel: route to sorting gate 1 regardless of destination *)
        SortingGate1 := TRUE;
        SortingGate2 := FALSE;
    ELSIF DestinationCodeSensor = 1 THEN
        (* Small parcel destined for Location A: route to sorting gate 2 *)
        SortingGate1 := FALSE;
        SortingGate2 := TRUE;
    ELSE
        (* Small parcel destined for Location B: keep on main conveyor *)
        SortingGate1 := FALSE;
        SortingGate2 := FALSE;
    END_IF;
ELSE
    (* Invalid parcel detected: stop conveyor and close all gates for safety *)
    ConveyorBeltMotor := FALSE;
    SortingGate1 := FALSE;
    SortingGate2 := FALSE;
END_IF;

END_FUNCTION_BLOCK

(* ---- med_85.st ---- *)
FUNCTION_BLOCK ShredderControl
VAR_INPUT
    StartButton : BOOL;         (* Momentary start button *)
    StopButton : BOOL;          (* Momentary stop button *)
    EmergencyStop : BOOL;       (* Emergency stop button - active high *)
    MaterialInFeed : BOOL;      (* Sensor detecting material at infeed *)
    JammedSensor : BOOL;        (* Sensor detecting jam condition - active high *)
END_VAR
VAR_OUTPUT
    MotorControl : BOOL;        (* Control signal to motor starter *)
    SafetyRelay : BOOL;         (* Safety relay control *)
END_VAR
VAR
    bMotorRunning : BOOL;       (* Internal motor running state *)
    bSafetyCondition : BOOL;    (* Internal safety status *)
END_VAR

(* 1. Safety Logic - Highest Priority *)
(* Emergency stop OR jam detection deactivates safety *)
bSafetyCondition := NOT EmergencyStop AND NOT JammedSensor;
SafetyRelay := bSafetyCondition;

(* 2. Motor Control Logic *)
IF bSafetyCondition THEN
    (* Normal operation allowed *)

    (* Start conditions:
       1. Start button pressed (momentary)
       2. Material detected at infeed (auto-start) *)
    IF StartButton OR MaterialInFeed THEN
        bMotorRunning := TRUE;
    END_IF;

    (* Stop condition: Stop button pressed (momentary) *)
    IF StopButton THEN
        bMotorRunning := FALSE;
    END_IF;

    (* Apply motor command *)
    MotorControl := bMotorRunning;
ELSE
    (* Safety override: Emergency stop or jam detected *)
    MotorControl := FALSE;
    bMotorRunning := FALSE;
END_IF;

END_FUNCTION_BLOCK

(* ---- med_86.st ---- *)
FUNCTION_BLOCK FruitJuicingBottling
VAR_INPUT
    StartButton : BOOL;        (* Input for starting the process *)
    StopButton : BOOL;         (* Input for stopping the process *)
    FruitSelected : BOOL;      (* Input indicating fruit selection *)
END_VAR
VAR_OUTPUT
    JuiceProcessing : BOOL;    (* Output for controlling juice extraction *)
    BottleFilling : BOOL;      (* Output for controlling bottle filling *)
    CapPlacement : BOOL;       (* Output for placing caps on bottles *)
    Packaging : BOOL;          (* Output for packaging filled bottles *)
    ProcessInProgress : BOOL;  (* Indicator for an ongoing process *)
END_VAR
VAR
    eState : (IDLE, RUNNING);  (* State variable for process control *)
END_VAR

(* Main process logic *)
CASE eState OF
    IDLE:
        (* Reset all outputs when idle *)
        ProcessInProgress := FALSE;
        JuiceProcessing := FALSE;
        BottleFilling := FALSE;
        CapPlacement := FALSE;
        Packaging := FALSE;

        (* Check start conditions: StartButton pressed, fruit selected, and no process running *)
        IF StartButton AND FruitSelected AND NOT ProcessInProgress THEN
            eState := RUNNING;
        END_IF;

    RUNNING:
        (* Set process indicator and activate all concurrent stages *)
        ProcessInProgress := TRUE;
        JuiceProcessing := TRUE;
        BottleFilling := TRUE;
        CapPlacement := TRUE;
        Packaging := TRUE;

        (* Check stop conditions: StopButton pressed OR fruit deselected *)
        IF StopButton OR NOT FruitSelected THEN
            eState := IDLE;
        END_IF;
END_CASE;
END_FUNCTION_BLOCK

(* ---- med_87.st ---- *)
FUNCTION_BLOCK WaterDesalination
VAR_INPUT
    StartButton : BOOL;          (* Input for starting the desalination process *)
    StopButton : BOOL;           (* Input for stopping the desalination process *)
    SalinitySensor : REAL;       (* Input for salinity level measurement *)
END_VAR
VAR_OUTPUT
    SeawaterInletValve : BOOL;   (* Output for seawater inlet valve control *)
    FreshwaterOutletValve : BOOL; (* Output for freshwater outlet valve control *)
    DesalinationInProgress : BOOL; (* Indicator for an ongoing desalination process *)
END_VAR
VAR
    MaxSalinity : REAL := 35.0;  (* Maximum allowable salinity in ppm for freshwater *)
    SalinityControlSeconds : INT := 0; (* Timer for salinity control in seconds *)
END_VAR

(* Main logic *)
IF StopButton THEN
    (* Stop process immediately when StopButton is pressed *)
    DesalinationInProgress := FALSE;
    SeawaterInletValve := FALSE;
    FreshwaterOutletValve := FALSE;
    SalinityControlSeconds := 0;
ELSIF StartButton AND NOT DesalinationInProgress THEN
    (* Start process when StartButton is pressed and process is not already running *)
    DesalinationInProgress := TRUE;
    SeawaterInletValve := TRUE;
    FreshwaterOutletValve := TRUE;
    SalinityControlSeconds := 0;
END_IF;

(* Salinity monitoring and control *)
IF DesalinationInProgress THEN
    (* Increment timer each scan cycle - assuming 1 second per cycle *)
    SalinityControlSeconds := SalinityControlSeconds + 1;

    (* Check salinity every 10 seconds *)
    IF SalinityControlSeconds >= 10 THEN
        IF SalinitySensor > MaxSalinity THEN
            (* Close freshwater outlet valve if salinity is too high *)
            FreshwaterOutletValve := FALSE;
        ELSE
            (* Keep freshwater outlet valve open if salinity is acceptable *)
            FreshwaterOutletValve := TRUE;
        END_IF;
        (* Reset timer after check *)
        SalinityControlSeconds := 0;
    END_IF;
END_IF;

END_FUNCTION_BLOCK

(* ---- med_88.st ---- *)
FUNCTION_BLOCK SmartLockerControl
VAR_INPUT
    AccessCode : INT;     (* User entered access code *)
    LockerNumber : INT;   (* Selected locker number (1-10) *)
END_VAR
VAR_OUTPUT
    LockerOpen : BOOL;    (* TRUE when locker should open *)
END_VAR
VAR
    LockerStatus : ARRAY[1..10] OF BOOL;      (* TRUE=occupied/locked, FALSE=empty/unlocked *)
    LockerAccessCode : ARRAY[1..10] OF INT;   (* Unique access codes for each locker *)
    bInitDone : BOOL;                         (* Initialization flag *)
    i : INT;                                  (* Loop counter for initialization *)
END_VAR

(* Initialization - runs only once *)
IF NOT bInitDone THEN
    (* Initialize all lockers to occupied/locked (TRUE) *)
    FOR i := 1 TO 10 DO
        LockerStatus[i] := TRUE;
    END_FOR;

    (* Set individual access codes for each locker *)
    LockerAccessCode[1] := 1234;
    LockerAccessCode[2] := 5678;
    LockerAccessCode[3] := 9876;
    LockerAccessCode[4] := 4321;
    LockerAccessCode[5] := 6543;
    LockerAccessCode[6] := 7890;
    LockerAccessCode[7] := 3456;
    LockerAccessCode[8] := 8765;
    LockerAccessCode[9] := 2345;
    LockerAccessCode[10] := 6789;

    bInitDone := TRUE;
END_IF;

(* Default output state *)
LockerOpen := FALSE;

(* Access control logic *)
IF (LockerNumber >= 1) AND (LockerNumber <= 10) THEN
    (* Check if access code matches and locker is currently locked *)
    IF (AccessCode = LockerAccessCode[LockerNumber]) AND LockerStatus[LockerNumber] THEN
        LockerOpen := TRUE;               (* Open the locker *)
        LockerStatus[LockerNumber] := FALSE; (* Mark as empty/unlocked *)
    END_IF;
END_IF;
END_FUNCTION_BLOCK

(* ---- med_89.st ---- *)
FUNCTION_BLOCK SoilTestingDeviceControl
VAR_INPUT
    StartButton : BOOL;           (* Input for starting the testing process *)
    SoilSampleDetected : BOOL;    (* Input for detecting soil sample *)
END_VAR

VAR_OUTPUT
    NutrientPump : BOOL;          (* Output to control nutrient pump *)
    pHAdjustmentPump : BOOL;      (* Output to control pH adjustment pump *)
END_VAR

VAR
    pHSensorValue : REAL;         (* Simulated pH sensor value *)
    NutrientSensorValue : REAL;   (* Simulated nutrient sensor value *)
    TestingStatus : INT;          (* Status: 0=Idle, 1=Testing, 2=Completed *)
    NutrientThreshold : REAL := 0.7;   (* Nutrient level threshold for analysis *)
    pHThreshold : REAL := 6.5;         (* pH level threshold for analysis *)
END_VAR

(* Main logic implementation *)
CASE TestingStatus OF
    0: (* Idle state *)
        (* Initialize sensor values *)
        pHSensorValue := 7.0;
        NutrientSensorValue := 0.5;

        (* Ensure pumps are off in idle state *)
        NutrientPump := FALSE;
        pHAdjustmentPump := FALSE;

        (* Check for start command *)
        IF StartButton THEN
            TestingStatus := 1;
            NutrientPump := TRUE;
            pHAdjustmentPump := TRUE;
        END_IF;

    1: (* Testing state *)
        (* Update simulated sensor values during testing *)
        IF NutrientSensorValue < 0.9 THEN
            NutrientSensorValue := NutrientSensorValue + 0.1;
        END_IF;

        IF pHSensorValue > 4.0 THEN
            pHSensorValue := pHSensorValue - 0.5;
        END_IF;

        (* Check for sample detection and analysis *)
        IF SoilSampleDetected THEN
            IF (NutrientSensorValue >= NutrientThreshold) AND (pHSensorValue <= pHThreshold) THEN
                TestingStatus := 2;
                NutrientPump := FALSE;
                pHAdjustmentPump := FALSE;
            END_IF;
        END_IF;

    2: (* Completed state *)
        (* Ensure pumps are off when testing is completed *)
        NutrientPump := FALSE;
        pHAdjustmentPump := FALSE;

        (* Optionally, the system could be reset to idle here if needed *)
        (* TestingStatus := 0; *)  (* Uncomment if automatic reset is desired *)
END_CASE;

END_FUNCTION_BLOCK

(* ---- med_90.st ---- *)
FUNCTION_BLOCK SushiConveyorControl
VAR_INPUT
    StartButton : BOOL;     (* Input to start the conveyor *)
    StopButton : BOOL;      (* Input to stop the conveyor *)
    EmergencyStop : BOOL;   (* Input for emergency stop *)
END_VAR
VAR_OUTPUT
    ConveyorMotor : BOOL;   (* Output to control the conveyor motor *)
END_VAR
VAR
    BeltRunning : BOOL;     (* Status of the conveyor: Running or Stopped *)
    ConveyorTimer : INT;    (* Timer counter for conveyor rotation *)
    RotationTime : INT := 5; (* Time for one rotation in seconds *)
END_VAR

(* Emergency Stop - Highest Priority *)
IF EmergencyStop THEN
    ConveyorMotor := FALSE;
    BeltRunning := FALSE;
    ConveyorTimer := 0;
    RETURN;
END_IF;

(* Start/Stop Control *)
IF StartButton AND NOT BeltRunning THEN
    ConveyorMotor := TRUE;
    BeltRunning := TRUE;
    ConveyorTimer := 0;
ELSIF StopButton AND BeltRunning THEN
    ConveyorMotor := FALSE;
    BeltRunning := FALSE;
    ConveyorTimer := 0;
END_IF;

(* Simulated Rotation Cycle *)
IF BeltRunning THEN
    ConveyorTimer := ConveyorTimer + 1;
    IF ConveyorTimer >= RotationTime THEN
        ConveyorTimer := 0;
    END_IF;
    ConveyorMotor := TRUE;
END_IF;

END_FUNCTION_BLOCK

(* ---- med_91.st ---- *)
FUNCTION_BLOCK AGVControlSystem
VAR_INPUT
    MaterialRequest : INT; (* 新的物料请求，>0表示有效请求 *)
    TaskComplete_AGV1 : BOOL := FALSE; (* AGV1任务完成信号 *)
    TaskComplete_AGV2 : BOOL := FALSE; (* AGV2任务完成信号 *)
    TaskComplete_AGV3 : BOOL := FALSE; (* AGV3任务完成信号 *)
    AGV1_PositionUpdate : INT := 0; (* AGV1位置更新值 *)
    AGV2_PositionUpdate : INT := 0; (* AGV2位置更新值 *)
    AGV3_PositionUpdate : INT := 0; (* AGV3位置更新值 *)
END_VAR

VAR_OUTPUT
    AGV1_Ready : BOOL := TRUE; (* AGV1就绪状态 *)
    AGV2_Ready : BOOL := TRUE; (* AGV2就绪状态 *)
    AGV3_Ready : BOOL := TRUE; (* AGV3就绪状态 *)
    AGV1_CurrentTask : INT := 0; (* AGV1当前任务，0表示空闲 *)
    AGV2_CurrentTask : INT := 0; (* AGV2当前任务，0表示空闲 *)
    AGV3_CurrentTask : INT := 0; (* AGV3当前任务，0表示空闲 *)
    AGV1_Position : INT := 0; (* AGV1当前位置 *)
    AGV2_Position : INT := 0; (* AGV2当前位置 *)
    AGV3_Position : INT := 0; (* AGV3当前位置 *)
    QueueCount : INT := 0; (* 队列中任务数量 *)
    SafetyError : BOOL := FALSE; (* 安全错误标志 *)
    QueueOverflow : BOOL := FALSE; (* 队列溢出标志 *)
    InvalidRequest : BOOL := FALSE; (* 无效请求标志 *)
END_VAR

VAR
    (* 物料处理请求队列 - FIFO实现 *)
    MaterialQueue : ARRAY[1..10] OF INT;
    QueueHead : INT := 1; (* 队列头部指针 *)
    QueueTail : INT := 1; (* 队列尾部指针 *)

    (* AGV状态管理 *)
    AGVStatus : ARRAY[1..3] OF BOOL := [TRUE, TRUE, TRUE]; (* TRUE=就绪，FALSE=工作中 *)
    AGVTask : ARRAY[1..3] OF INT := [0, 0, 0]; (* AGV当前任务 *)

    (* 临时变量 *)
    TempTask : INT;
    i : INT;

    (* 状态监控 *)
    PreviousQueueCount : INT := 0;
    SystemIdle : BOOL := TRUE;
END_VAR

(* 1. 处理新的物料请求 *)
InvalidRequest := FALSE;
IF MaterialRequest > 0 THEN
    (* 检查请求有效性 *)
    IF MaterialRequest <= 100 THEN  (* 假设有效任务ID范围1-100 *)
        IF QueueCount < 10 THEN
            (* 原子性队列更新 *)
            MaterialQueue[QueueTail] := MaterialRequest;
            QueueTail := QueueTail + 1;
            IF QueueTail > 10 THEN
                QueueTail := 1;
            END_IF;
            QueueCount := QueueCount + 1;
            QueueOverflow := FALSE;
        ELSE
            (* 队列溢出处理 *)
            QueueOverflow := TRUE;
            SafetyError := TRUE;
        END_IF;
    ELSE
        (* 无效请求处理 *)
        InvalidRequest := TRUE;
        SafetyError := TRUE;
    END_IF;
END_IF;

(* 2. 处理AGV任务完成 *)
(* AGV1任务完成处理 *)
IF TaskComplete_AGV1 AND NOT AGVStatus[1] THEN
    AGVStatus[1] := TRUE;
    AGVTask[1] := 0;
    AGV1_Position := 0; (* 重置位置 *)
END_IF;

(* AGV2任务完成处理 *)
IF TaskComplete_AGV2 AND NOT AGVStatus[2] THEN
    AGVStatus[2] := TRUE;
    AGVTask[2] := 0;
    AGV2_Position := 0; (* 重置位置 *)
END_IF;

(* AGV3任务完成处理 *)
IF TaskComplete_AGV3 AND NOT AGVStatus[3] THEN
    AGVStatus[3] := TRUE;
    AGVTask[3] := 0;
    AGV3_Position := 0; (* 重置位置 *)
END_IF;

(* 3. 优先级任务分配策略 *)
IF QueueCount > 0 THEN
    (* 从队列头部获取任务 *)
    TempTask := MaterialQueue[QueueHead];

    (* 优先级分配：AGV1 > AGV2 > AGV3 *)
    IF AGVStatus[1] THEN
        (* 分配任务给AGV1 *)
        AGVTask[1] := TempTask;
        AGVStatus[1] := FALSE;

        (* 更新队列 *)
        QueueHead := QueueHead + 1;
        IF QueueHead > 10 THEN
            QueueHead := 1;
        END_IF;
        QueueCount := QueueCount - 1;

    ELSIF AGVStatus[2] THEN
        (* 分配任务给AGV2 *)
        AGVTask[2] := TempTask;
        AGVStatus[2] := FALSE;

        (* 更新队列 *)
        QueueHead := QueueHead + 1;
        IF QueueHead > 10 THEN
            QueueHead := 1;
        END_IF;
        QueueCount := QueueCount - 1;

    ELSIF AGVStatus[3] THEN
        (* 分配任务给AGV3 *)
        AGVTask[3] := TempTask;
        AGVStatus[3] := FALSE;

        (* 更新队列 *)
        QueueHead := QueueHead + 1;
        IF QueueHead > 10 THEN
            QueueHead := 1;
        END_IF;
        QueueCount := QueueCount - 1;
    END_IF;
END_IF;

(* 4. 更新AGV位置并实施安全约束 *)
(* AGV1位置更新 *)
IF NOT AGVStatus[1] THEN
    AGV1_Position := AGV1_Position + AGV1_PositionUpdate;
    (* 安全约束：确保位置非负 *)
    IF AGV1_Position < 0 THEN
        AGV1_Position := 0;
        SafetyError := TRUE;
    END_IF;
END_IF;

(* AGV2位置更新 *)
IF NOT AGVStatus[2] THEN
    AGV2_Position := AGV2_Position + AGV2_PositionUpdate;
    (* 安全约束：确保位置非负 *)
    IF AGV2_Position < 0 THEN
        AGV2_Position := 0;
        SafetyError := TRUE;
    END_IF;
END_IF;

(* AGV3位置更新 *)
IF NOT AGVStatus[3] THEN
    AGV3_Position := AGV3_Position + AGV3_PositionUpdate;
    (* 安全约束：确保位置非负 *)
    IF AGV3_Position < 0 THEN
        AGV3_Position := 0;
        SafetyError := TRUE;
    END_IF;
END_IF;

(* 5. 状态监控和同步 *)
(* 更新输出状态 *)
AGV1_Ready := AGVStatus[1];
AGV2_Ready := AGVStatus[2];
AGV3_Ready := AGVStatus[3];

AGV1_CurrentTask := AGVTask[1];
AGV2_CurrentTask := AGVTask[2];
AGV3_CurrentTask := AGVTask[3];

(* 监控系统空闲状态 *)
SystemIdle := (QueueCount = 0) AND AGVStatus[1] AND AGVStatus[2] AND AGVStatus[3];

(* 监控状态转换一致性 *)
IF PreviousQueueCount > QueueCount AND QueueCount > 0 THEN
    (* 队列任务减少但未分配任务，检查状态一致性 *)
    IF AGVStatus[1] AND AGVStatus[2] AND AGVStatus[3] THEN
        SafetyError := TRUE; (* 所有AGV就绪但队列任务减少，状态不一致 *)
    END_IF;
END_IF;
PreviousQueueCount := QueueCount;

(* 6. 错误处理恢复机制 *)
(* 如果系统空闲且无错误，清除安全错误标志 *)
IF SystemIdle AND NOT QueueOverflow AND NOT InvalidRequest THEN
    SafetyError := FALSE;
END_IF;

(* 确保任务不会重复分配 *)
FOR i := 1 TO 3 DO
    IF AGVTask[i] <> 0 THEN
        (* 检查其他AGV是否有相同任务 *)
        IF (i = 1 AND (AGVTask[2] = AGVTask[1] OR AGVTask[3] = AGVTask[1])) OR
           (i = 2 AND (AGVTask[1] = AGVTask[2] OR AGVTask[3] = AGVTask[2])) OR
           (i = 3 AND (AGVTask[1] = AGVTask[3] OR AGVTask[2] = AGVTask[3])) THEN
            SafetyError := TRUE;
            (* 重置重复的任务 *)
            IF i = 1 THEN AGVTask[1] := 0; AGVStatus[1] := TRUE; END_IF;
            IF i = 2 THEN AGVTask[2] := 0; AGVStatus[2] := TRUE; END_IF;
            IF i = 3 THEN AGVTask[3] := 0; AGVStatus[3] := TRUE; END_IF;
        END_IF;
    END_IF;
END_FOR;

END_FUNCTION_BLOCK
